{attribute 'GeneratedUsingTerminal: KL9191'}
{attribute addProperty BoxType "KL9191"}
{attribute addProperty Id "Channel_1AT %Q*Channel_471FAA5C0"}
{attribute addProperty CRC "2519344351"}
{attribute addProperty Size "0"}
TYPE KL9191_962A24DF :
STRUCT
	{attribute addProperty Name "Channel_1"}
	Channel_1 : Channel_471FAA5C;
END_STRUCT
END_TYPE

(* stored: Version 1.2.0.0, ProductVersion 3.1.4024.9
   DUT KL9191_962A24DF: Id {78008f2a-f9b4-4043-8d50-f74a7ed31243} *)
